//-----------------------------------------------------------------------------------------
//
//                  			ST_HMI_Transfer_ArmCnc
//
//						Structure HMI transfert entre bras et cnc		
//-----------------------------------------------------------------------------------------
//
//Auteur: G.GOETZ
//Création: 20.02.2026
//Dernière modification : 20.02.2026 (G.GOETZ)
//       			
//-----------------------------------------------------------------------------------------
//
//     							Liste des modifications  	
//
// 20.02.2026 (G.GOETZ) -> Création		
//-----------------------------------------------------------------------------------------

TYPE ST_HMI_Transfer_ArmCnc :
STRUCT

	(** SETUP FLAG **)
		(*Arm*)
			bCheckSensorArmGripper1 : BOOL ; // Check the sensor of the arm gripper 1
			bCheckSensorArmGripper2 : BOOL ; // Check the sensor of the arm gripper 2

END_STRUCT
END_TYPE

(* stored: Version 1.1.0.1, ProductVersion 3.1.4026.17
   DUT ST_HMI_Transfer_ArmCnc: Id {14044221-30b0-47eb-b32e-de72ed179a91} *)
